INTERFACE I_Testsuite EXTENDS I_Base

PROPERTY PUBLIC P_File : String(255)
GET
END_GET
SET
END_SET
END_PROPERTY

PROPERTY PUBLIC P_List : I_ListSTRING
GET
END_GET
END_PROPERTY

PROPERTY PUBLIC P_Logger : I_Logger
GET
END_GET
SET
END_SET
END_PROPERTY

PROPERTY PUBLIC P_Options : reference to ST_TestsuiteOptions
GET
END_GET
END_PROPERTY

PROPERTY PUBLIC P_Parent : I_Testsuites
GET
END_GET
SET
END_SET
END_PROPERTY

PROPERTY PUBLIC P_Testcase : INT
GET
END_GET
END_PROPERTY

END_INTERFACE

(* stored: Version 1.1.0.1
   Itf I_Testsuite: Id {be1b8503-88c7-00d0-316f-5b2753f7b610}
   Property P_File: Id {a818bff5-ba3d-0c59-3d5e-9f25ce58cd33}
   Get Get: Id {cedd11f8-8c12-0ca0-3de4-d95b3ccb4746}
   Set Set: Id {4cc4cce7-b779-00b2-3ed3-bcd8149eb033}
   Property P_List: Id {8c44755e-2744-0f94-1f92-c5697833051a}
   Get Get: Id {1f7d7b47-83e0-07fc-1005-a59bd3ef5268}
   Property P_Logger: Id {ed5121df-8a75-0b78-2403-edba980ee298}
   Get Get: Id {332f727d-4af8-0dcd-3c33-20e0c188cc99}
   Set Set: Id {48759934-cc6c-0535-18d0-64ac77c2d5c5}
   Property P_Options: Id {95855609-76ef-038e-19f4-6cb57a551cda}
   Get Get: Id {66a90f66-147e-08b8-06bc-16760d564648}
   Property P_Parent: Id {dec8515c-cb5f-06f1-34a8-4435601bd530}
   Get Get: Id {bf712599-e9a4-0d4b-2139-f66f32ed9d3c}
   Set Set: Id {a60365dc-68ca-0323-3ca8-1abefc7debdb}
   Property P_Testcase: Id {4e4b87c6-fedd-0eea-3a95-04aa9817daa1}
   Get Get: Id {e80fe4c8-79ad-0f5d-03c0-493d759378fe} *)
